// TwinCAT 3 PLC project StepperTest
// ProgramVersion: 3.1.4023.0
// libraries:
//   MqttFramework, * (FactoryAutomation)
//   StateMachineLib, * (FactoryAutomation)
//   Tc2_MC2, * (Beckhoff Automation GmbH)
//   Tc2_Standard, * (Beckhoff Automation GmbH)
//   Tc2_System, * (Beckhoff Automation GmbH)
//   Tc3_Module, * (Beckhoff Automation GmbH)
//   VisuSymbols,3.5.10.0,System
// project tree:
//   / GlobalTextList.TcGTLO, PlcTask.TcTTO, Visualisierungsmanager.TcVMO (not stored)
//   POUs/ MAIN.TcPOU
//   POUs/Motion/ Axis.TcPOU, I_Axis.TcIO
//   VISUs/ fAxis.TcVIS, Visualization.TcVIS
// real-time tasks:
//   TASK PlcTask: cycle T#10ms, priority 20, ADS port 350
// motion (NC):
//   TASK NC-Task 1 SAF: cycle T#6ms, priority 4, ADS port 501
//   TASK NC-Task 1 SVB: cycle T#10ms, priority 8, ADS port 511
//   AXIS Achse P (id 1)
//     OtherSettings: AllowMotionCmdToSlave=true
//     encoder EncType=1
//       Inc: RefSearchInverse=true, RefSyncInverse=false, RefSoftSyncMask=#x0000ffff
//     drive DrvType=24
//       Analog: TorqueSetpointScale=10, ScaleFactorActTorque=0.1
//       TimeComp: TaskDelayCycles=1
//     controller CtrType=1
//       CtrPara: PriorControlFactor=1
//         Observer: BandWidth=20
//   AXIS Achse X (id 2)
//     Dynamic: Acceleration=1525.5, Deceleration=1525.5, Jerk=1989.02
//     Velo: RefSearch=3, RefSync=1, SlowManual=1, FastManual=10, Maximum=350
//     OtherSettings: AllowMotionCmdToSlave=true
//     encoder EncType=4
//       EncPara: ScaleFactorNumerator=0.0799, ScaleFactorDenominator=25, EncMode=1, MaxCount=#x0000ffff
//         SoftEndMinControl: Enable=true
//         SoftEndMaxControl: Enable=true, Range=300
//         Inc: RefSearchInverse=true, RefSyncInverse=false, RefMode=1, RefSoftSyncMask=#x0000ffff
//     drive DrvType=24
//       Analog: VeloReferenz=400, TorqueSetpointScale=10, ScaleFactorActTorque=0.1
//       TimeComp: TaskDelayCycles=1
//     controller CtrType=1
//       CtrPara: PriorControlFactor=1
//         PosDiffControl: Enable=false
//         Observer: BandWidth=20
//   AXIS Achse Y (id 3)
//     Velo: Maximum=9000
//     OtherSettings: AllowMotionCmdToSlave=true
//     encoder EncType=1
//       Inc: RefSoftSyncMask=#x0000ffff
//     drive DrvType=24
//       Analog: VeloReferenz=400, TorqueSetpointScale=10, ScaleFactorActTorque=0.1
//       TimeComp: TaskDelayCycles=1
//     controller CtrType=1
//       CtrPara: PriorControlFactor=1
//         Observer: BandWidth=20
//   AXIS Achse Z1 (id 4)
//     OtherSettings: AllowMotionCmdToSlave=true
//     encoder EncType=1
//       Inc: RefSoftSyncMask=#x0000ffff
//     drive DrvType=24
//       Analog: TorqueSetpointScale=10, ScaleFactorActTorque=0.1
//       TimeComp: TaskDelayCycles=1
//     controller CtrType=1
//       CtrPara: PriorControlFactor=1
//         Observer: BandWidth=20
//   AXIS Achse Z2 (id 5)
//     OtherSettings: AllowMotionCmdToSlave=true
//     encoder EncType=1
//       Inc: RefSoftSyncMask=#x0000ffff
//     drive DrvType=24
//       Analog: TorqueSetpointScale=10, ScaleFactorActTorque=0.1
//       TimeComp: TaskDelayCycles=1
//     controller CtrType=1
//       CtrPara: PriorControlFactor=1
//         Observer: BandWidth=20
// I/O:
//   DEVICE Gerät 3 (EtherCAT), AmsNetId 192.168.56.1.4.1
//     Klemme 1 (EK1100) [EK1100 EtherCAT-Koppler (2A E-Bus)]
//       Klemme 12 (EL7031) [EL7031 1K. Schrittmotor-Endstufe (24V, 1.5A)]
//       Klemme 3 (EL7031) [EL7031 1K. Schrittmotor-Endstufe (24V, 1.5A)]
//       Klemme 4 (EL7031) [EL7031 1K. Schrittmotor-Endstufe (24V, 1.5A)]
//       Klemme 5 (EL7031) [EL7031 1K. Schrittmotor-Endstufe (24V, 1.5A)]
//       Klemme 6 (EL7031) [EL7031 1K. Schrittmotor-Endstufe (24V, 1.5A)]
//       Klemme 7 (EL9011) [EL9011 Endklemme]
// variable links:
//   NC-Task 1 SAF/Axes/Achse P <-> Device 3 (EtherCAT)/Term 1 (EK1100)/Term 12 (EL7031)
//     Drive/Inputs/In/nState1 @bit 3 <-> STM Status/Status/Error
//     Drive/Inputs/In/nState1 @bit 5 <-> STM Status/Status/Moving negative
//     Drive/Inputs/In/nState1 @bit 4 <-> STM Status/Status/Moving positive
//     Drive/Inputs/In/nState1 @bit 1 <-> STM Status/Status/Ready
//     Drive/Inputs/In/nState1 <-> STM Status/Status/Ready to enable
//     Drive/Inputs/In/nState1 @bit 6 <-> STM Status/Status/Torque reduced
//     Drive/Inputs/In/nState1 @bit 2 <-> STM Status/Status/Warning
//     Drive/Inputs/In/nState2 @bit 3 <-> STM Status/Status/Digital input 1
//     Drive/Inputs/In/nState2 @bit 4 <-> STM Status/Status/Digital input 2
//     Drive/Inputs/In/nState4 @bit 1 <-> WcState/InputToggle
//     Drive/Inputs/In/nState4 <-> WcState/WcState
//     Drive/Outputs/Out/nCtrl1 <-> STM Control/Control/Enable
//     Drive/Outputs/Out/nCtrl1 @bit 2 <-> STM Control/Control/Reduce torque
//     Drive/Outputs/Out/nCtrl1 @bit 1 <-> STM Control/Control/Reset
//     Drive/Outputs/Out/nDataOut2[0] <-> STM Velocity/Velocity
//     Enc/Inputs/In/nDataIn1[0] <-> ENC Status compact/Counter value
//     Enc/Inputs/In/nDataIn2[0] <-> ENC Status compact/Latch value
//     Enc/Inputs/In/nState1 @bit 4 <-> ENC Status compact/Status/Counter overflow
//     Enc/Inputs/In/nState1 @bit 3 <-> ENC Status compact/Status/Counter underflow
//     Enc/Inputs/In/nState1 @bit 1 <-> ENC Status compact/Status/Latch extern valid
//     Enc/Inputs/In/nState1 @bit 2 <-> ENC Status compact/Status/Set counter done
//     Enc/Inputs/In/nState2 @bit 4 <-> ENC Status compact/Status/Status of extern latch
//     Enc/Inputs/In/nState4 @bit 1 <-> WcState/InputToggle
//     Enc/Inputs/In/nState4 <-> WcState/WcState
//     Enc/Outputs/Out/nCtrl1 @bit 3 <-> ENC Control compact/Control/Enable latch extern on negative edge
//     Enc/Outputs/Out/nCtrl1 @bit 1 <-> ENC Control compact/Control/Enable latch extern on positive edge
//     Enc/Outputs/Out/nCtrl1 @bit 2 <-> ENC Control compact/Control/Set counter
//     Enc/Outputs/Out/nDataOut1[0] <-> ENC Control compact/Set counter value
//   NC-Task 1 SAF/Axes/Achse X <-> Device 3 (EtherCAT)/Term 1 (EK1100)/Term 3 (EL7031)
//     Drive/Inputs/In/nState1 @bit 3 <-> STM Status/Status/Error
//     Drive/Inputs/In/nState1 @bit 5 <-> STM Status/Status/Moving negative
//     Drive/Inputs/In/nState1 @bit 4 <-> STM Status/Status/Moving positive
//     Drive/Inputs/In/nState1 @bit 1 <-> STM Status/Status/Ready
//     Drive/Inputs/In/nState1 <-> STM Status/Status/Ready to enable
//     Drive/Inputs/In/nState1 @bit 6 <-> STM Status/Status/Torque reduced
//     Drive/Inputs/In/nState1 @bit 2 <-> STM Status/Status/Warning
//     Drive/Inputs/In/nState4 @bit 1 <-> WcState/InputToggle
//     Drive/Inputs/In/nState4 <-> WcState/WcState
//     Drive/Outputs/Out/nCtrl1 <-> STM Control/Control/Enable
//     Drive/Outputs/Out/nCtrl1 @bit 2 <-> STM Control/Control/Reduce torque
//     Drive/Outputs/Out/nCtrl1 @bit 1 <-> STM Control/Control/Reset
//     Drive/Outputs/Out/nDataOut2[0] <-> STM Velocity/Velocity
//     Enc/Inputs/In/nDataIn1[0] <-> ENC Status compact/Counter value
//     Enc/Inputs/In/nDataIn2[0] <-> ENC Status compact/Latch value
//     Enc/Inputs/In/nState1 @bit 4 <-> ENC Status compact/Status/Counter overflow
//     Enc/Inputs/In/nState1 @bit 3 <-> ENC Status compact/Status/Counter underflow
//     Enc/Inputs/In/nState1 @bit 1 <-> ENC Status compact/Status/Latch extern valid
//     Enc/Inputs/In/nState1 @bit 2 <-> ENC Status compact/Status/Set counter done
//     Enc/Inputs/In/nState2 @bit 4 <-> ENC Status compact/Status/Status of extern latch
//     Enc/Inputs/In/nState4 @bit 1 <-> WcState/InputToggle
//     Enc/Inputs/In/nState4 <-> WcState/WcState
//     Enc/Outputs/Out/nCtrl1 @bit 3 <-> ENC Control compact/Control/Enable latch extern on negative edge
//     Enc/Outputs/Out/nCtrl1 @bit 1 <-> ENC Control compact/Control/Enable latch extern on positive edge
//     Enc/Outputs/Out/nCtrl1 @bit 2 <-> ENC Control compact/Control/Set counter
//     Enc/Outputs/Out/nDataOut1[0] <-> ENC Control compact/Set counter value
//   NC-Task 1 SAF/Axes/Achse Y <-> Device 3 (EtherCAT)/Term 1 (EK1100)/Term 4 (EL7031)
//     Drive/Inputs/In/nState1 @bit 3 <-> STM Status/Status/Error
//     Drive/Inputs/In/nState1 @bit 5 <-> STM Status/Status/Moving negative
//     Drive/Inputs/In/nState1 @bit 4 <-> STM Status/Status/Moving positive
//     Drive/Inputs/In/nState1 @bit 1 <-> STM Status/Status/Ready
//     Drive/Inputs/In/nState1 <-> STM Status/Status/Ready to enable
//     Drive/Inputs/In/nState1 @bit 6 <-> STM Status/Status/Torque reduced
//     Drive/Inputs/In/nState1 @bit 2 <-> STM Status/Status/Warning
//     Drive/Inputs/In/nState2 @bit 5 <-> STM Status/Status/Sync error
//     Drive/Inputs/In/nState2 @bit 7 <-> STM Status/Status/TxPDO Toggle
//     Drive/Inputs/In/nState4 @bit 1 <-> WcState/InputToggle
//     Drive/Inputs/In/nState4 <-> WcState/WcState
//     Drive/Outputs/Out/nCtrl1 <-> STM Control/Control/Enable
//     Drive/Outputs/Out/nCtrl1 @bit 2 <-> STM Control/Control/Reduce torque
//     Drive/Outputs/Out/nCtrl1 @bit 1 <-> STM Control/Control/Reset
//     Drive/Outputs/Out/nDataOut2[0] <-> STM Velocity/Velocity
//     Enc/Inputs/In/nDataIn1[0] <-> ENC Status compact/Counter value
//     Enc/Inputs/In/nDataIn2[0] <-> ENC Status compact/Latch value
//     Enc/Inputs/In/nState1 @bit 4 <-> ENC Status compact/Status/Counter overflow
//     Enc/Inputs/In/nState1 @bit 3 <-> ENC Status compact/Status/Counter underflow
//     Enc/Inputs/In/nState1 @bit 1 <-> ENC Status compact/Status/Latch extern valid
//     Enc/Inputs/In/nState1 @bit 2 <-> ENC Status compact/Status/Set counter done
//     Enc/Inputs/In/nState2 @bit 4 <-> ENC Status compact/Status/Status of extern latch
//     Enc/Inputs/In/nState2 @bit 5 <-> ENC Status compact/Status/Sync error
//     Enc/Inputs/In/nState2 @bit 7 <-> ENC Status compact/Status/TxPDO Toggle
//     Enc/Inputs/In/nState4 @bit 1 <-> WcState/InputToggle
//     Enc/Inputs/In/nState4 <-> WcState/WcState
//     Enc/Outputs/Out/nCtrl1 @bit 3 <-> ENC Control compact/Control/Enable latch extern on negative edge
//     Enc/Outputs/Out/nCtrl1 @bit 1 <-> ENC Control compact/Control/Enable latch extern on positive edge
//     Enc/Outputs/Out/nCtrl1 @bit 2 <-> ENC Control compact/Control/Set counter
//     Enc/Outputs/Out/nDataOut1[0] <-> ENC Control compact/Set counter value
//   NC-Task 1 SAF/Axes/Achse Z1 <-> Device 3 (EtherCAT)/Term 1 (EK1100)/Term 5 (EL7031)
//     Drive/Inputs/In/nState1 @bit 3 <-> STM Status/Status/Error
//     Drive/Inputs/In/nState1 @bit 5 <-> STM Status/Status/Moving negative
//     Drive/Inputs/In/nState1 @bit 4 <-> STM Status/Status/Moving positive
//     Drive/Inputs/In/nState1 @bit 1 <-> STM Status/Status/Ready
//     Drive/Inputs/In/nState1 <-> STM Status/Status/Ready to enable
//     Drive/Inputs/In/nState1 @bit 6 <-> STM Status/Status/Torque reduced
//     Drive/Inputs/In/nState1 @bit 2 <-> STM Status/Status/Warning
//     Drive/Inputs/In/nState2 @bit 3 <-> STM Status/Status/Digital input 1
//     Drive/Inputs/In/nState2 @bit 4 <-> STM Status/Status/Digital input 2
//     Drive/Inputs/In/nState4 @bit 1 <-> WcState/InputToggle
//     Drive/Inputs/In/nState4 <-> WcState/WcState
//     Drive/Outputs/Out/nCtrl1 <-> STM Control/Control/Enable
//     Drive/Outputs/Out/nCtrl1 @bit 2 <-> STM Control/Control/Reduce torque
//     Drive/Outputs/Out/nCtrl1 @bit 1 <-> STM Control/Control/Reset
//     Drive/Outputs/Out/nDataOut2[0] <-> STM Velocity/Velocity
//     Enc/Inputs/In/nDataIn1[0] <-> ENC Status compact/Counter value
//     Enc/Inputs/In/nDataIn2[0] <-> ENC Status compact/Latch value
//     Enc/Inputs/In/nState1 @bit 4 <-> ENC Status compact/Status/Counter overflow
//     Enc/Inputs/In/nState1 @bit 3 <-> ENC Status compact/Status/Counter underflow
//     Enc/Inputs/In/nState1 @bit 1 <-> ENC Status compact/Status/Latch extern valid
//     Enc/Inputs/In/nState1 @bit 2 <-> ENC Status compact/Status/Set counter done
//     Enc/Inputs/In/nState2 @bit 4 <-> ENC Status compact/Status/Status of extern latch
//     Enc/Inputs/In/nState4 @bit 1 <-> WcState/InputToggle
//     Enc/Inputs/In/nState4 <-> WcState/WcState
//     Enc/Outputs/Out/nCtrl1 @bit 3 <-> ENC Control compact/Control/Enable latch extern on negative edge
//     Enc/Outputs/Out/nCtrl1 @bit 1 <-> ENC Control compact/Control/Enable latch extern on positive edge
//     Enc/Outputs/Out/nCtrl1 @bit 2 <-> ENC Control compact/Control/Set counter
//     Enc/Outputs/Out/nDataOut1[0] <-> ENC Control compact/Set counter value
//   NC-Task 1 SAF/Axes/Achse Z2 <-> Device 3 (EtherCAT)/Term 1 (EK1100)/Term 6 (EL7031)
//     Drive/Inputs/In/nState1 @bit 3 <-> STM Status/Status/Error
//     Drive/Inputs/In/nState1 @bit 5 <-> STM Status/Status/Moving negative
//     Drive/Inputs/In/nState1 @bit 4 <-> STM Status/Status/Moving positive
//     Drive/Inputs/In/nState1 @bit 1 <-> STM Status/Status/Ready
//     Drive/Inputs/In/nState1 <-> STM Status/Status/Ready to enable
//     Drive/Inputs/In/nState1 @bit 6 <-> STM Status/Status/Torque reduced
//     Drive/Inputs/In/nState1 @bit 2 <-> STM Status/Status/Warning
//     Drive/Inputs/In/nState2 @bit 3 <-> STM Status/Status/Digital input 1
//     Drive/Inputs/In/nState2 @bit 4 <-> STM Status/Status/Digital input 2
//     Drive/Inputs/In/nState4 @bit 1 <-> WcState/InputToggle
//     Drive/Inputs/In/nState4 <-> WcState/WcState
//     Drive/Outputs/Out/nCtrl1 <-> STM Control/Control/Enable
//     Drive/Outputs/Out/nCtrl1 @bit 2 <-> STM Control/Control/Reduce torque
//     Drive/Outputs/Out/nCtrl1 @bit 1 <-> STM Control/Control/Reset
//     Drive/Outputs/Out/nDataOut2[0] <-> STM Velocity/Velocity
//     Enc/Inputs/In/nDataIn1[0] <-> ENC Status compact/Counter value
//     Enc/Inputs/In/nDataIn2[0] <-> ENC Status compact/Latch value
//     Enc/Inputs/In/nState1 @bit 4 <-> ENC Status compact/Status/Counter overflow
//     Enc/Inputs/In/nState1 @bit 3 <-> ENC Status compact/Status/Counter underflow
//     Enc/Inputs/In/nState1 @bit 1 <-> ENC Status compact/Status/Latch extern valid
//     Enc/Inputs/In/nState1 @bit 2 <-> ENC Status compact/Status/Set counter done
//     Enc/Inputs/In/nState2 @bit 4 <-> ENC Status compact/Status/Status of extern latch
//     Enc/Inputs/In/nState4 @bit 1 <-> WcState/InputToggle
//     Enc/Inputs/In/nState4 <-> WcState/WcState
//     Enc/Outputs/Out/nCtrl1 @bit 3 <-> ENC Control compact/Control/Enable latch extern on negative edge
//     Enc/Outputs/Out/nCtrl1 @bit 1 <-> ENC Control compact/Control/Enable latch extern on positive edge
//     Enc/Outputs/Out/nCtrl1 @bit 2 <-> ENC Control compact/Control/Set counter
//     Enc/Outputs/Out/nDataOut1[0] <-> ENC Control compact/Set counter value
//   StepperTest/StepperTest Instance <-> Device 3 (EtherCAT)/Term 1 (EK1100)/Term 3 (EL7031)
//     PlcTask Inputs/MAIN.fbXAxis.bCalibrationCam <-> STM Status/Status/Digital input 1
//   StepperTest/StepperTest Instance <-> NC-Task 1 SAF/Axes/Achse X
//     PlcTask Inputs/MAIN.fbXAxis.axisRef.NcToPlc <-> Outputs/ToPlc
//     PlcTask Outputs/MAIN.fbXAxis.axisRef.PlcToNc <-> Inputs/FromPlc
//   StepperTest/StepperTest Instance <-> NC-Task 1 SAF/Axes/Achse Y
//     PlcTask Inputs/MAIN.fbYAxis.axisRef.NcToPlc <-> Outputs/ToPlc
//     PlcTask Outputs/MAIN.fbYAxis.axisRef.PlcToNc <-> Inputs/FromPlc

CONFIGURATION StepperTest
    RESOURCE PLC ON TwinCAT3
        TASK PlcTask(INTERVAL := T#10ms, PRIORITY := 20);
        PROGRAM MAIN WITH PlcTask : MAIN;
        PROGRAM ADS WITH PlcTask : ADS;
    END_RESOURCE
END_CONFIGURATION

// ---- POUs/Motion/I_Axis.TcIO
INTERFACE I_Axis

METHOD PrepareDecoupling : I_Axis
VAR_INPUT
	slaveAxis : REFERENCE TO AXIS_REF;
	slaveStatus : REFERENCE TO ST_AXISSTATUS;
END_VAR
END_METHOD

METHOD StartCoupling : I_Axis
VAR_INPUT
END_VAR
END_METHOD

METHOD StartDecoupling : BOOL
VAR_INPUT
END_VAR
END_METHOD

METHOD StartHoming : BOOL;
VAR_INPUT
END_VAR
END_METHOD

END_INTERFACE

// ---- POUs/MAIN.TcPOU
PROGRAM MAIN
VAR
	fbXAxis : Axis;
	fbYAxis : Axis;
	fbZ1Axis : Axis;
	fbZ2Axis : Axis;
	
	bHomeZ1Z2Axis : BOOL;
	bHomeXYAxis : BOOL;
	bHomingStarted : BOOL;
	bDecoupleXYAxis : BOOL;
	diStep : DINT;
	sTLMqttName: STRING(8) := 'PLC_CHAN';
	messageIndex: UINT;
	stMqttPayload: MqttFramework.ST_MqttPayload;
	sMessage : STRING;
	evalIndex : INT;
END_VAR

fbXAxis();
fbYAxis();

IF bDecoupleXYAxis
THEN

	IF fbXAxis
		.PrepareDecoupling(fbYAxis.axisRef,fbYAxis.fbMcReadStatus.Status)
		.StartDecoupling()
	THEN
		//Decoupling successful
		bDecoupleXYAxis := FALSE;
	END_IF
	
END_IF

IF bHomeXYAxis
THEN
	
	IF fbXAxis
		.PrepareCoupling(fbYAxis.axisRef,fbYAxis.fbMcReadStatus.Status, -1, 1)
		.StartCoupling()
		.StartHoming()
	THEN
		bHomeXYAxis := FALSE;
		bHomingStarted := FALSE;
	END_IF
	
END_IF


CASE diStep OF
	
	0:
	
		IF ADS.fbMqttClient.Subscribe(sTopic := sTLMqttName)
		THEN			
			diStep := 10;
		END_IF
	
	
	10:
	
		messageIndex := ADS.fbMqttClient.isNewMessage(sTLMqttName);
		IF messageIndex > 0
		THEN
			stMqttPayload := Ads.fbMqttClient.getNewMessage(messageIndex);
			diStep:=20;
		END_IF
		
	//Payloadauswertung	
	20:
	
		sMessage := '';
		FOR evalIndex := 1 TO 32 DO
			sMessage := CONCAT(sMessage , F_ToCHR(stMqttPayload.data[evalIndex]));
		END_FOR
		
		diStep:=30;
	
	30:
	
		IF sMessage = 'cmd_home'
		THEN
			bHomeXYAxis := TRUE;
			diStep := 10;
		END_IF
	
END_CASE

END_PROGRAM

// ---- POUs/Motion/Axis.TcPOU
FUNCTION_BLOCK Axis IMPLEMENTS I_AXIS
VAR_INPUT
	bEnable : BOOL;
	bHalt : BOOL;
	bStop : BOOL;
	bReset : BOOL;
END_VAR
VAR_OUTPUT
	axisRef : AXIS_REF;
	fbMcReadStatus : MC_ReadStatus;
END_VAR
VAR
	bCalibrationCam AT%I* :  BOOL;
	
	//Data for coupling operations
	//--------------------------------------------------------------
	
	slaveAxis : REFERENCE TO AXIS_REF;
	slaveStatus : REFERENCE TO ST_AXISSTATUS;
	lrRatioNumerator : LREAL := 1;
	uiRatioDenominator : UINT := 1;
	
	//--------------------------------------------------------------
	
	fbMcHome : MC_Home;
	fbMcGearIn : MC_GearIn;
	fbMcGearOut : MC_GearOut;
	
	fbMcPower : MC_Power;
	fbMcHalt : MC_Halt;
	fbMcStop : MC_Stop;
	fbMcReset : MC_Reset;
END_VAR

fbMcStop(
	Axis:= axisRef, 
	Execute:= bStop
);
	
fbMcHalt(
	Axis:= axisRef, 
	Execute:= bHalt
);
	
fbMcReset(
	Axis:= axisRef, 
	Execute:= bReset
);
	
fbMcPower(
	Axis:= axisRef, 
	Enable:= bEnable, 
	Enable_Positive:= bEnable, 
	Enable_Negative:= bEnable, 
	Override:= , 
	BufferMode:= , 
	Options:= , 
	Status=> , 
	Busy=> , 
	Active=> , 
	Error=> , 
	ErrorID=> 
);

fbMcReadStatus(
	Axis:= axisRef, 
	Enable:= TRUE, 
);

fbMcHome(
	Axis:= axisRef, 
	bCalibrationCam:= bCalibrationCam, 
);

IF 		__ISVALIDREF(slaveAxis)
	AND __ISVALIDREF(slaveStatus)
THEN

	fbMcGearIn(
		Master:= axisRef, 
		Slave:= slaveAxis, 
		RatioNumerator:= lrRatioNumerator, 
		RatioDenominator:= uiRatioDenominator
	);
	
	IF NOT fbMcGearIn.Busy
	THEN
		fbMcGearIn.Execute := FALSE;
	END_IF
	
	
	fbMcGearOut(Slave:= slaveAxis);
	IF NOT fbMcGearOut.Busy
	THEN
		fbMcGearOut.Execute := FALSE;
	END_IF
	
END_IF


IF fbMcHome.Done
THEN
	fbMcHome.Execute := FALSE;
END_IF

METHOD PrepareCoupling : I_Axis
VAR_INPUT
	slaveAxis : REFERENCE TO AXIS_REF;
	slaveStatus : REFERENCE TO ST_AXISSTATUS;
	lrRatioNumerator : LREAL;
	uiRatioDenominator : UINT;
END_VAR
PrepareCoupling := THIS^;
THIS^.slaveAxis REF= slaveAxis;
THIS^.slaveStatus REF= slaveStatus;
THIS^.lrRatioNumerator := lrRatioNumerator;
THIS^.uiRatioDenominator := uiRatioDenominator;
END_METHOD

METHOD PrepareDecoupling : I_Axis
VAR_INPUT
	slaveAxis : REFERENCE TO AXIS_REF;
	slaveStatus : REFERENCE TO ST_AXISSTATUS;
END_VAR
PrepareDecoupling := THIS^;
THIS^.slaveAxis REF= slaveAxis;
THIS^.slaveStatus REF= slaveStatus;
END_METHOD

METHOD StartCoupling : I_Axis
VAR_INPUT
END_VAR
StartCoupling := THIS^;
IF NOT __ISVALIDREF(slaveStatus)
THEN
	RETURN;
END_IF

IF NOT slaveStatus.Coupled
THEN
	fbMcGearIn.Execute := TRUE;
END_IF
END_METHOD

METHOD StartDecoupling : BOOL
VAR_INPUT
END_VAR

IF NOT __ISVALIDREF(slaveStatus)
THEN
	RETURN;
END_IF

IF slaveStatus.Coupled
THEN
	fbMcGearOut.Execute := TRUE;
ELSE
	StartDecoupling := TRUE;
END_IF
END_METHOD

METHOD StartHoming : BOOL;
VAR_INPUT
END_VAR
IF NOT fbMcGearIn.Execute
	//AND fbMcReadStatus.Valid
	//AND NOT fbMcReadStatus.Status.Homed 
THEN
	
	fbMcHome.Execute := TRUE;
	IF fbMcHome.Busy
	THEN
		fbMcHome.Execute := FALSE;
		StartHoming := TRUE;
	END_IF
	
END_IF
END_METHOD

END_FUNCTION_BLOCK

// ---- GlobalTextList.TcGTLO
TEXTLIST GlobalTextList
  293 = '%d'
  99 = 'Decouple XY Axis'
  16 = 'Enable'
  421 = 'Halt'
  472 = 'Home XY AXis'
  216 = 'Home XY Axis'
  355 = 'Reset'
  740 = 'Stop'
END_TEXTLIST

// ---- VISUs/fAxis.TcVIS
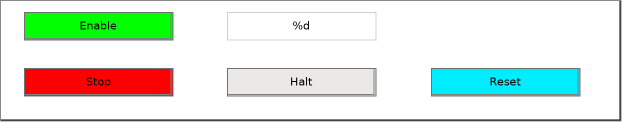
VISUALIZATION fAxis  // 622x122
VAR_IN_OUT
	io_fbAxis : Axis;
END_VAR
    Rectangle (0,0 620x120)
    Button (24,68 149x28), "Stop"
        tap io_fbAxis.bStop
    Textfield (227,12 149x28), "%d", text variable: io_fbAxis.axisRef.NcToPlc.AxisId
    Button (227,68 149x28), "Halt"
        tap io_fbAxis.bHalt
    Button (431,68 149x28), "Reset"
        tap io_fbAxis.bReset
    Button (24,12 149x28), "Enable"
        toggle io_fbAxis.bEnable
END_VISUALIZATION

// ---- VISUs/Visualization.TcVIS
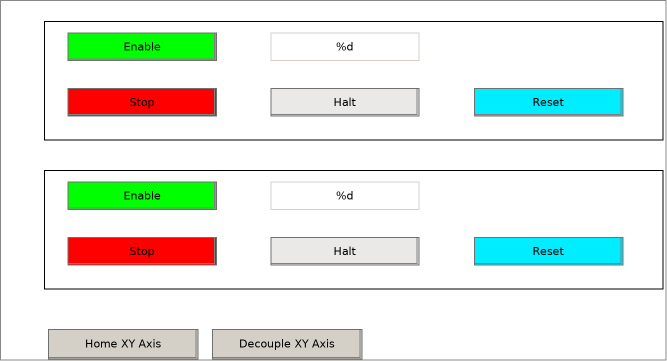
VISUALIZATION Visualization  // 667x361
    Frame (44,21 621x121)
        shows fAxis(io_fbAxis := MAIN.fbXAxis)
    Frame (44,170 621x121)
        shows fAxis(io_fbAxis := MAIN.fbYAxis)
    Button (48,329 150x30), "Home XY Axis"
        toggle MAIN.bHomeXYAxis
    Button (212,329 150x30), "Decouple XY Axis"
        toggle MAIN.bDecoupleXYAxis
END_VISUALIZATION
